Omron CX-Programmer project NewProject (CX-Programmer 9.70)

# PLC NewPLC1: CP1L M

## Global symbols (name address type ; comment)
0.00 BOOL  ; Glass
0.01 BOOL  ; Plastic
0.02 BOOL  ; SW_Done
0.03 BOOL  ; SW_RESET
0.04 BOOL  ; Reset Technician
0.05 BOOL  ; SW_DONOR
0.06 BOOL  ; Cal
0.07 BOOL  ; Can
0.10 BOOL  ; reset
0.11 BOOL  ; plastic limit
0.12 BOOL  ; Glass limit
0.13 BOOL  ; Can limit
100.00 BOOL  ; Conveyor 1
100.01 BOOL  ; Conveyor 2
100.02 BOOL  ; RETURN BOTTOM
100.03 BOOL  ; Storage G
100.04 BOOL  ; Storage P
100.05 BOOL  ; Storage C
100.06 BOOL  ; Conveyor 3
101.00 BOOL  ; Glass Limit
102.00 BOOL  ; Plastic Limit
103.00 BOOL  ; Can limit
1.00 BOOL  ; SW_COKE
1.01 BOOL  ; SW_SNACKs
1.02 BOOL  ; SW_WATER
1.03 BOOL  ; SW_CANDY
200.00 BOOL  ; LED COKE.
200.01 BOOL  ; LED SNACKs
200.02 BOOL  ; LED WATER
200.03 BOOL  ; LED CANDY
D0 CHANNEL  ; Path1
D1 CHANNEL  ; Path2
D100 CHANNEL  ; GP
D101 CHANNEL  ; PP
D102 CHANNEL  ; CP
D4 CHANNEL  ; Bottlescore1
D5 CHANNEL  ; Bottlescore2
D6 CHANNEL  ; TotalBottles
D7 CHANNEL  ; TotalUser
D8 CHANNEL  ; Path 3
P PointU
PM PointM
PU PointM
PointM PointU
PointUSer PointM

## Program NewProgram1 (cyclic task 0)

### Section Section1

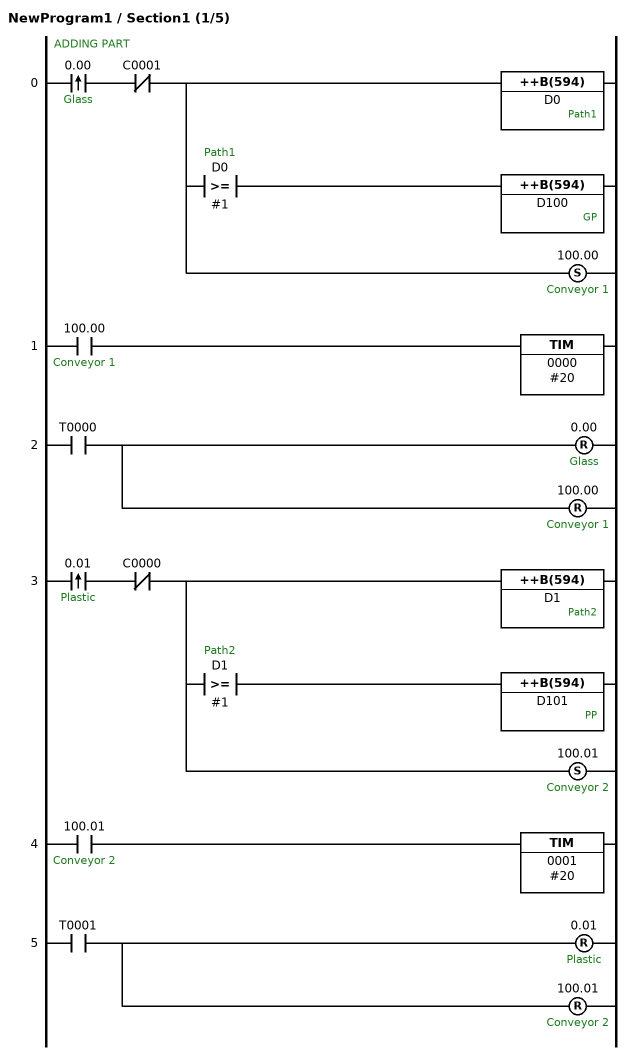
; rung 0: ADDING PART
@LD 0.00  ; Glass
ANDNOT C0001
OUT TR0
++B(594) D0  ; Path1
AND>=(325) D0 #1  ; Path1
++B(594) D100  ; GP
LD TR0
SET 100.00  ; Conveyor 1
; rung 1
LD 100.00  ; Conveyor 1
TIM 0000 #20
; rung 2
LD T0000
RSET 0.00  ; Glass
RSET 100.00  ; Conveyor 1
; rung 3
@LD 0.01  ; Plastic
ANDNOT C0000
OUT TR0
++B(594) D1  ; Path2
AND>=(325) D1 #1  ; Path2
++B(594) D101  ; PP
LD TR0
SET 100.01  ; Conveyor 2
; rung 4
LD 100.01  ; Conveyor 2
TIM 0001 #20
; rung 5
LD T0001
RSET 0.01  ; Plastic
RSET 100.01  ; Conveyor 2

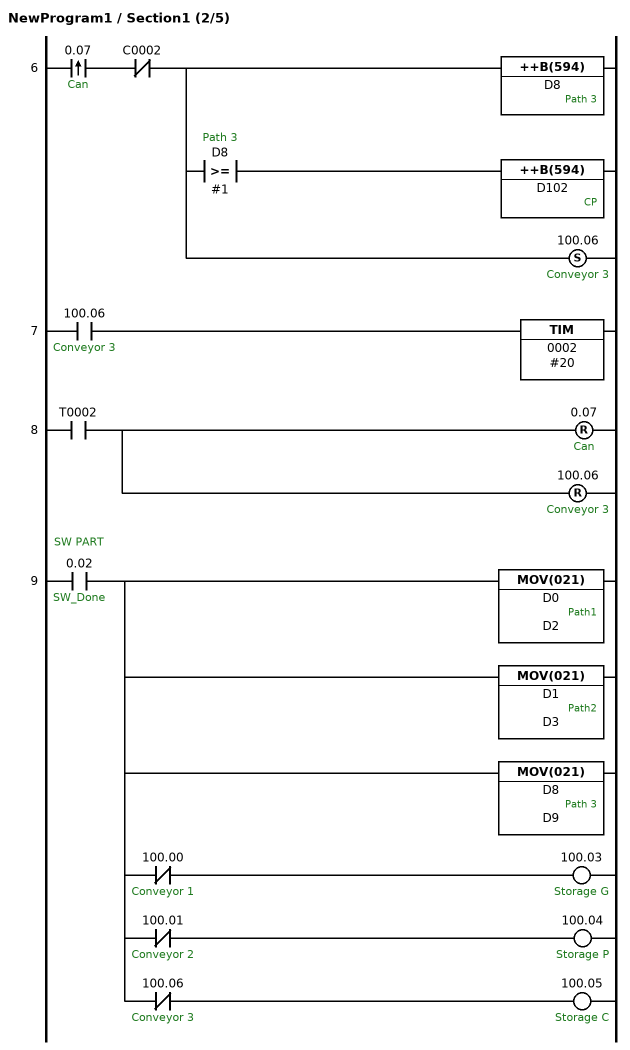
; rung 6
@LD 0.07  ; Can
ANDNOT C0002
OUT TR0
++B(594) D8  ; Path 3
AND>=(325) D8 #1  ; Path 3
++B(594) D102  ; CP
LD TR0
SET 100.06  ; Conveyor 3
; rung 7
LD 100.06  ; Conveyor 3
TIM 0002 #20
; rung 8
LD T0002
RSET 0.07  ; Can
RSET 100.06  ; Conveyor 3
; rung 9: SW PART
LD 0.02  ; SW_Done
OUT TR0
MOV(021) D0 D2  ; Path1
MOV(021) D1 D3  ; Path2
MOV(021) D8 D9  ; Path 3
ANDNOT 100.00  ; Conveyor 1
OUT 100.03  ; Storage G
LD TR0
ANDNOT 100.01  ; Conveyor 2
OUT 100.04  ; Storage P
LD TR0
ANDNOT 100.06  ; Conveyor 3
OUT 100.05  ; Storage C

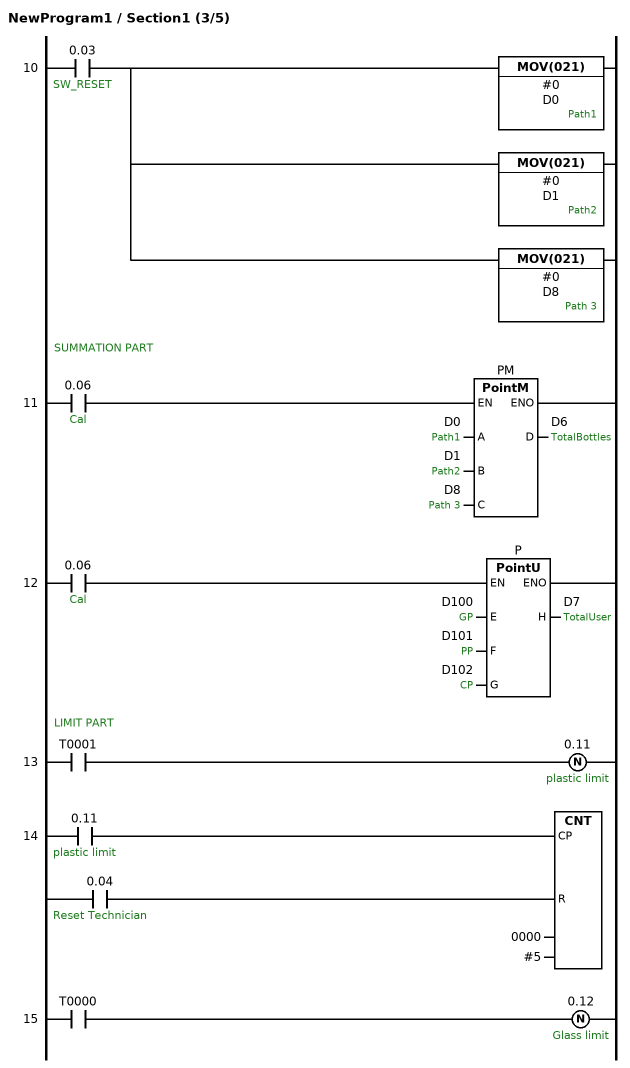
; rung 10
LD 0.03  ; SW_RESET
MOV(021) #0 D0  ; Path1
MOV(021) #0 D1  ; Path2
MOV(021) #0 D8  ; Path 3
; rung 11: SUMMATION PART
LD 0.06  ; Cal
CALL PM : PointM (A := D0, B := D1, C := D8, D => D6)  ; Path1, Path2, Path 3, TotalBottles
; rung 12
LD 0.06  ; Cal
CALL P : PointU (E := D100, F := D101, G := D102, H => D7)  ; GP, PP, CP, TotalUser
; rung 13: LIMIT PART
LD T0001
DIFD(014) 0.11  ; plastic limit
; rung 14
LD 0.11  ; plastic limit
LD 0.04  ; Reset Technician
CNT 0000 #5
; rung 15
LD T0000
DIFD(014) 0.12  ; Glass limit

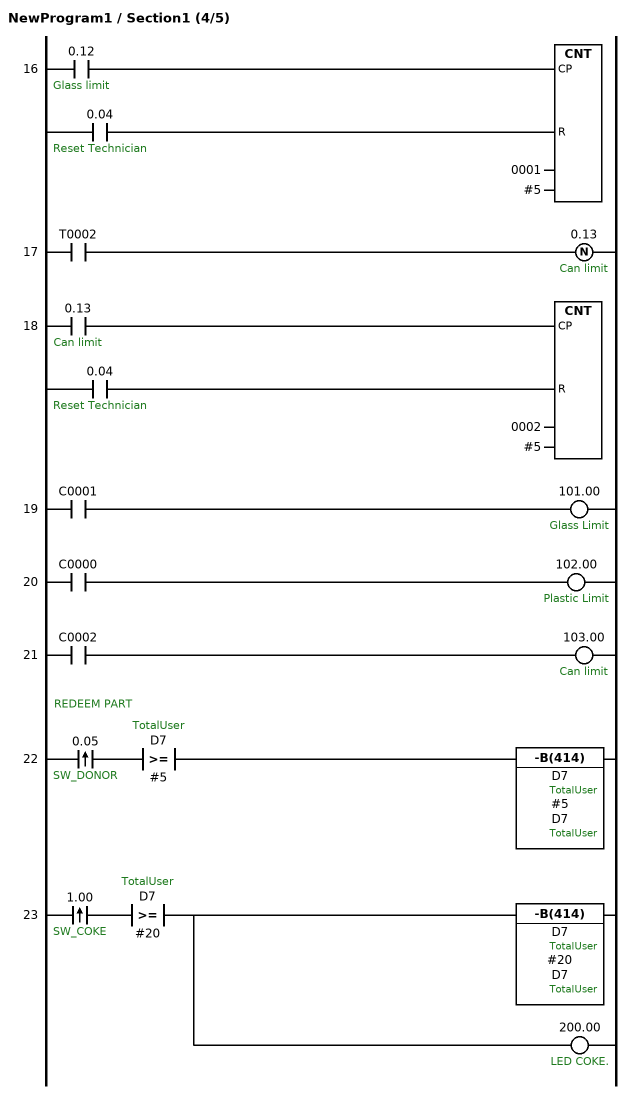
; rung 16
LD 0.12  ; Glass limit
LD 0.04  ; Reset Technician
CNT 0001 #5
; rung 17
LD T0002
DIFD(014) 0.13  ; Can limit
; rung 18
LD 0.13  ; Can limit
LD 0.04  ; Reset Technician
CNT 0002 #5
; rung 19
LD C0001
OUT 101.00  ; Glass Limit
; rung 20
LD C0000
OUT 102.00  ; Plastic Limit
; rung 21
LD C0002
OUT 103.00  ; Can limit
; rung 22: REDEEM PART
@LD 0.05  ; SW_DONOR
AND>=(325) D7 #5  ; TotalUser
-B(414) D7 #5 D7  ; TotalUser
; rung 23
@LD 1.00  ; SW_COKE
AND>=(325) D7 #20  ; TotalUser
-B(414) D7 #20 D7  ; TotalUser
OUT 200.00  ; LED COKE.

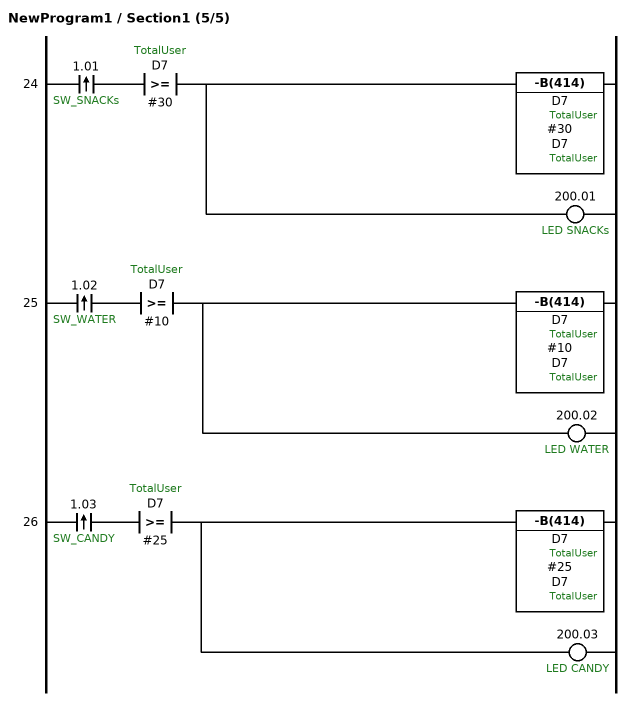
; rung 24
@LD 1.01  ; SW_SNACKs
AND>=(325) D7 #30  ; TotalUser
-B(414) D7 #30 D7  ; TotalUser
OUT 200.01  ; LED SNACKs
; rung 25
@LD 1.02  ; SW_WATER
AND>=(325) D7 #10  ; TotalUser
-B(414) D7 #10 D7  ; TotalUser
OUT 200.02  ; LED WATER
; rung 26
@LD 1.03  ; SW_CANDY
AND>=(325) D7 #25  ; TotalUser
-B(414) D7 #25 D7  ; TotalUser
OUT 200.03  ; LED CANDY

### Section END
; rung 0
END(001)

## Function block PointM
VAR_INPUT
  A : INT;
  B : INT;
  C : INT;
END_VAR
VAR_OUTPUT
  D : INT;
END_VAR
D  := A + B +C ;

## Function block PointU
VAR_INPUT
  E : INT;
  F : INT;
  G : INT;
END_VAR
VAR_OUTPUT
  H : INT;
END_VAR
	H := E + F + G;